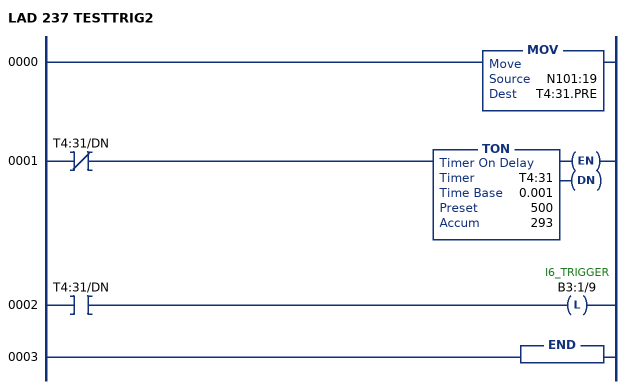
% Rung: 0 %
SOR MOV N101:19 T4:31.PRE EOR
%   N101:19  I6_TRIGTIME  "test trgiger 6 interval" %
% Rung: 1 %
SOR XIO T4:31/DN TON T4:31 0.001 500 293 EOR
% Rung: 2 %
SOR XIC T4:31/DN OTL B3:1/9 EOR
%   B3:1/9  I6_TRIGGER %
% Rung: 3 %
SOR END EOR

LADDER 238 "TESTTRIG3"
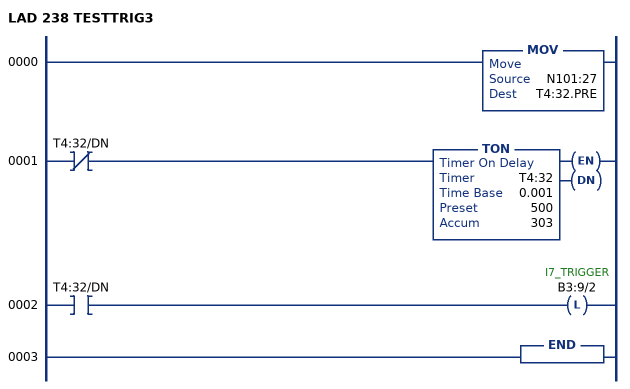
% Rung: 0 %
SOR MOV N101:27 T4:32.PRE EOR
%   N101:27  I7_TRIGTIME %
% Rung: 1 %
SOR XIO T4:32/DN TON T4:32 0.001 500 303 EOR
% Rung: 2 %
SOR XIC T4:32/DN OTL B3:9/2 EOR
%   B3:9/2  I7_TRIGGER %
% Rung: 3 %
SOR END EOR

LADDER 239 "TESTTRIG4"
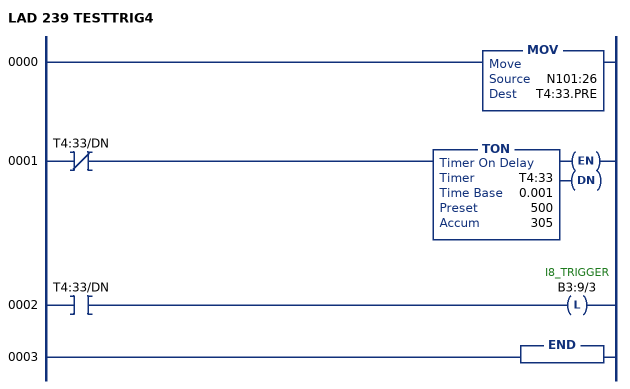
% Rung: 0 %
SOR MOV N101:26 T4:33.PRE EOR
%   N101:26  I8_TRIGTIME %
% Rung: 1 %
SOR XIO T4:33/DN TON T4:33 0.001 500 305 EOR
% Rung: 2 %
SOR XIC T4:33/DN OTL B3:9/3 EOR
%   B3:9/3  I8_TRIGGER %
% Rung: 3 %
SOR END EOR

LADDER 240 "TESTTRIG5"
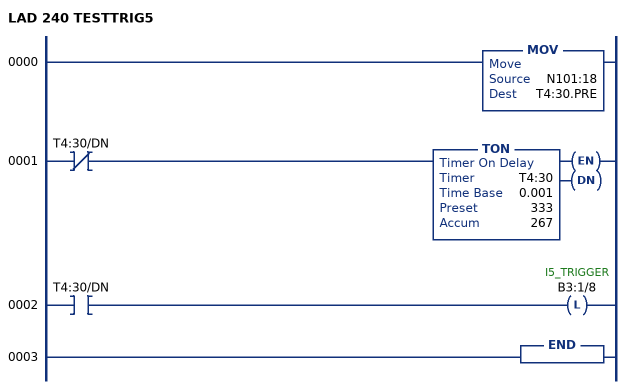
% Rung: 0 %
SOR MOV N101:18 T4:30.PRE EOR
%   N101:18  I5_TRIGTIME  "test trigger 5 interval" %
% Rung: 1 %
SOR XIO T4:30/DN TON T4:30 0.001 333 267 EOR
% Rung: 2 %
SOR XIC T4:30/DN OTL B3:1/8 EOR
%   B3:1/8  I5_TRIGGER %
% Rung: 3 %
SOR END EOR

LADDER 241 "TESTTRIG6"
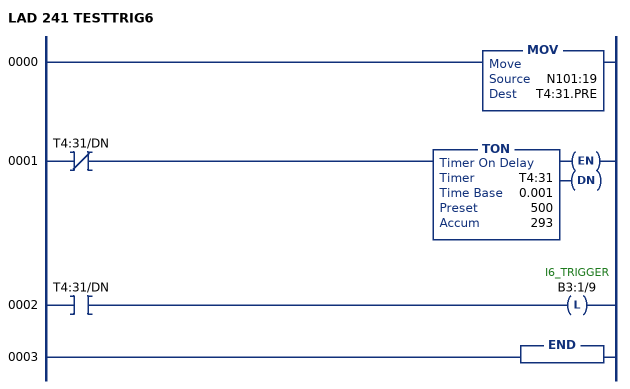
% Rung: 0 %
SOR MOV N101:19 T4:31.PRE EOR
%   N101:19  I6_TRIGTIME  "test trgiger 6 interval" %
% Rung: 1 %
SOR XIO T4:31/DN TON T4:31 0.001 500 293 EOR
% Rung: 2 %
SOR XIC T4:31/DN OTL B3:1/9 EOR
%   B3:1/9  I6_TRIGGER %
% Rung: 3 %
SOR END EOR

LADDER 242 "TESTTRIG7"
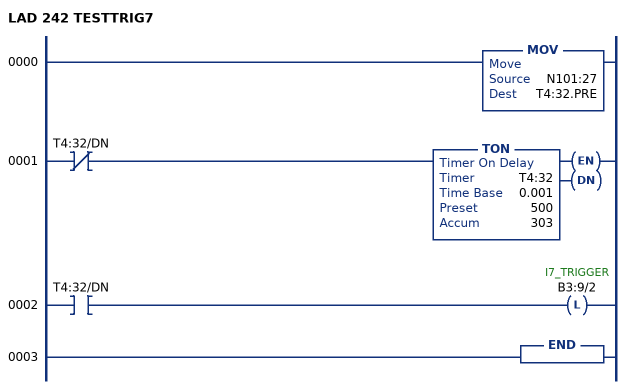
% Rung: 0 %
SOR MOV N101:27 T4:32.PRE EOR
%   N101:27  I7_TRIGTIME %
% Rung: 1 %
SOR XIO T4:32/DN TON T4:32 0.001 500 303 EOR
% Rung: 2 %
SOR XIC T4:32/DN OTL B3:9/2 EOR
%   B3:9/2  I7_TRIGGER %
% Rung: 3 %
SOR END EOR

LADDER 243 "TESTTRIG8"
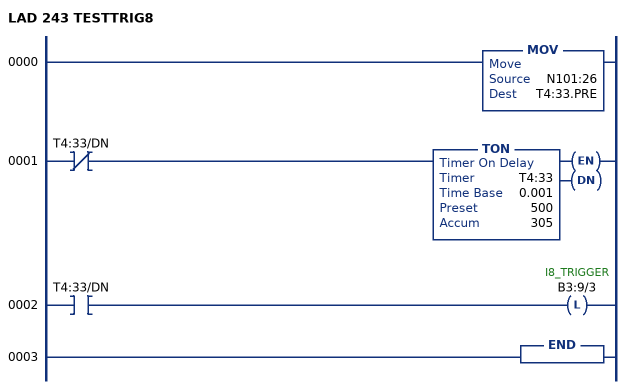
% Rung: 0 %
SOR MOV N101:26 T4:33.PRE EOR
%   N101:26  I8_TRIGTIME %
% Rung: 1 %
SOR XIO T4:33/DN TON T4:33 0.001 500 305 EOR
% Rung: 2 %
SOR XIC T4:33/DN OTL B3:9/3 EOR
%   B3:9/3  I8_TRIGGER %
% Rung: 3 %
SOR END EOR

LADDER 244 "PACKAGER"    % normal %
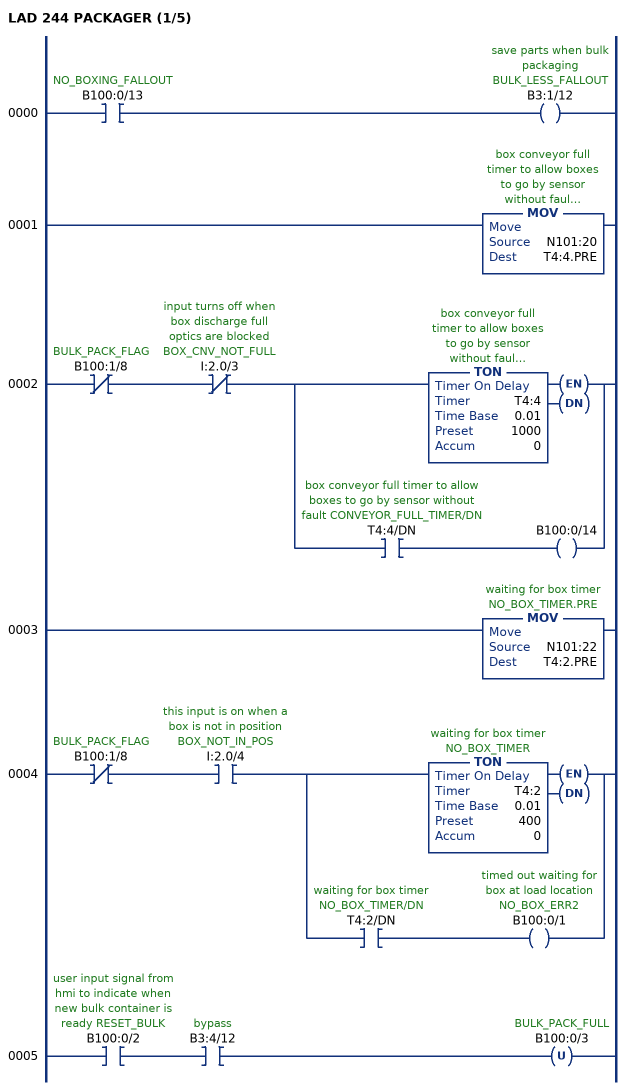
% Rung: 0 %
SOR XIC B100:0/13 OTE B3:1/12 EOR
%   B100:0/13  NO_BOXING_FALLOUT %
%   B3:1/12  BULK_LESS_FALLOUT  "save parts when bulk packaging" %
% Rung: 1 %
SOR MOV N101:20 T4:4.PRE EOR
%   N101:20  CONV_FULL_TIME_LIMIT  "time to allow box to pass box conveyor full sensor without fault" %
%   T4:4  CONVEYOR_FULL_TIMER  "box conveyor full timer to allow boxes to go by sensor without fault" %
% Rung: 2 %
SOR XIO B100:1/8 XIO I:2.0/3 BST TON T4:4 0.01 1000 0 NXB XIC T4:4/DN OTE B100:0/14 BND EOR
%   B100:1/8  BULK_PACK_FLAG %
%   I:2.0/3  BOX_CNV_NOT_FULL  "input turns off when box discharge full optics are blocked" %
%   T4:4  CONVEYOR_FULL_TIMER  "box conveyor full timer to allow boxes to go by sensor without fault" %
% Rung: 3 %
SOR MOV N101:22 T4:2.PRE EOR
%   N101:22  BOX_WAIT_TIME_LIMIT  "the time until waiting for box message in hmi (fault)" %
%   T4:2  NO_BOX_TIMER  "waiting for box timer" %
% Rung: 4 %
SOR XIO B100:1/8 XIC I:2.0/4 BST TON T4:2 0.01 400 0 NXB XIC T4:2/DN OTE B100:0/1 BND EOR
%   B100:1/8  BULK_PACK_FLAG %
%   I:2.0/4  BOX_NOT_IN_POS  "this input is on when a box is not in position" %
%   T4:2  NO_BOX_TIMER  "waiting for box timer" %
%   B100:0/1  NO_BOX_ERR2  "timed out waiting for box at load location" %
% Rung: 5 %
SOR XIC B100:0/2 XIC B3:4/12 OTU B100:0/3 EOR
%   B100:0/2  RESET_BULK  "user input signal from hmi to indicate when new bulk container is ready" %
%   B3:4/12  "bypass" %
%   B100:0/3  BULK_PACK_FULL %

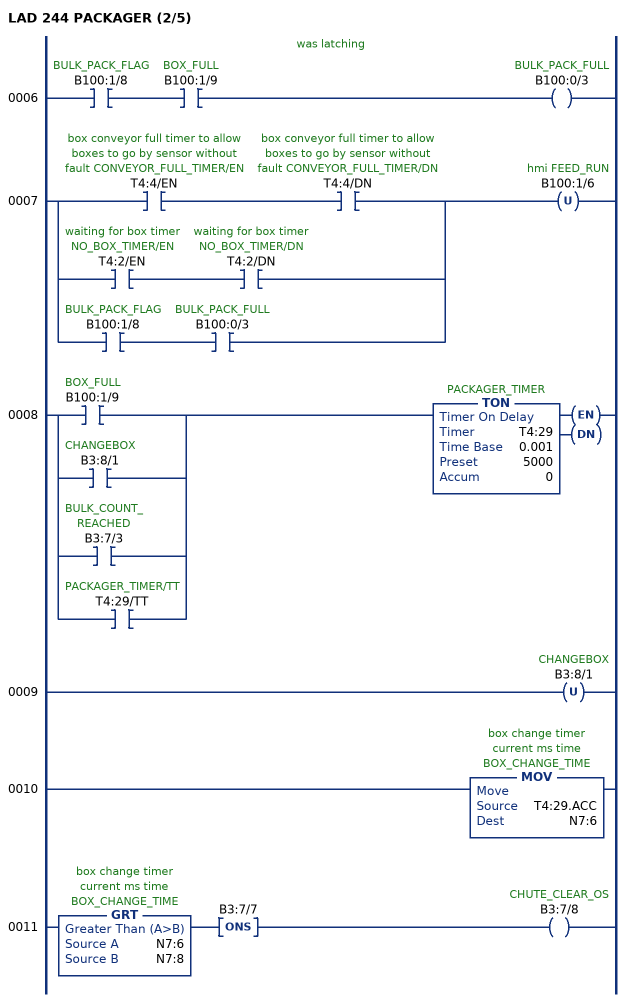
% Rung: 6 %
% was latching %
SOR XIC B100:1/8 XIC B100:1/9 OTE B100:0/3 EOR
%   B100:1/8  BULK_PACK_FLAG %
%   B100:1/9  BOX_FULL %
%   B100:0/3  BULK_PACK_FULL %
% Rung: 7 %
SOR BST XIC T4:4/EN XIC T4:4/DN NXB XIC T4:2/EN XIC T4:2/DN NXB XIC B100:1/8 XIC B100:0/3 BND OTU B100:1/6 EOR
%   T4:4  CONVEYOR_FULL_TIMER  "box conveyor full timer to allow boxes to go by sensor without fault" %
%   T4:2  NO_BOX_TIMER  "waiting for box timer" %
%   B100:1/8  BULK_PACK_FLAG %
%   B100:0/3  BULK_PACK_FULL %
%   B100:1/6  FEED_RUN  "hmi" %
% Rung: 8 %
SOR BST XIC B100:1/9 NXB XIC B3:8/1 NXB XIC B3:7/3 NXB XIC T4:29/TT BND TON T4:29 0.001 5000 0 EOR
%   B100:1/9  BOX_FULL %
%   B3:8/1  CHANGEBOX %
%   B3:7/3  BULK_COUNT_REACHED %
%   T4:29  PACKAGER_TIMER %
% Rung: 9 %
SOR OTU B3:8/1 EOR
%   B3:8/1  CHANGEBOX %
% Rung: 10 %
SOR MOV T4:29.ACC N7:6 EOR
%   T4:29  PACKAGER_TIMER %
%   N7:6  BOX_CHANGE_TIME  "box change timer current ms time" %
% Rung: 11 %
SOR GRT N7:6 N7:8 ONS B3:7/7 OTE B3:7/8 EOR
%   N7:6  BOX_CHANGE_TIME  "box change timer current ms time" %
%   N7:8  CHUTE_CLEAR_TIME %
%   B3:7/8  CHUTE_CLEAR_OS %

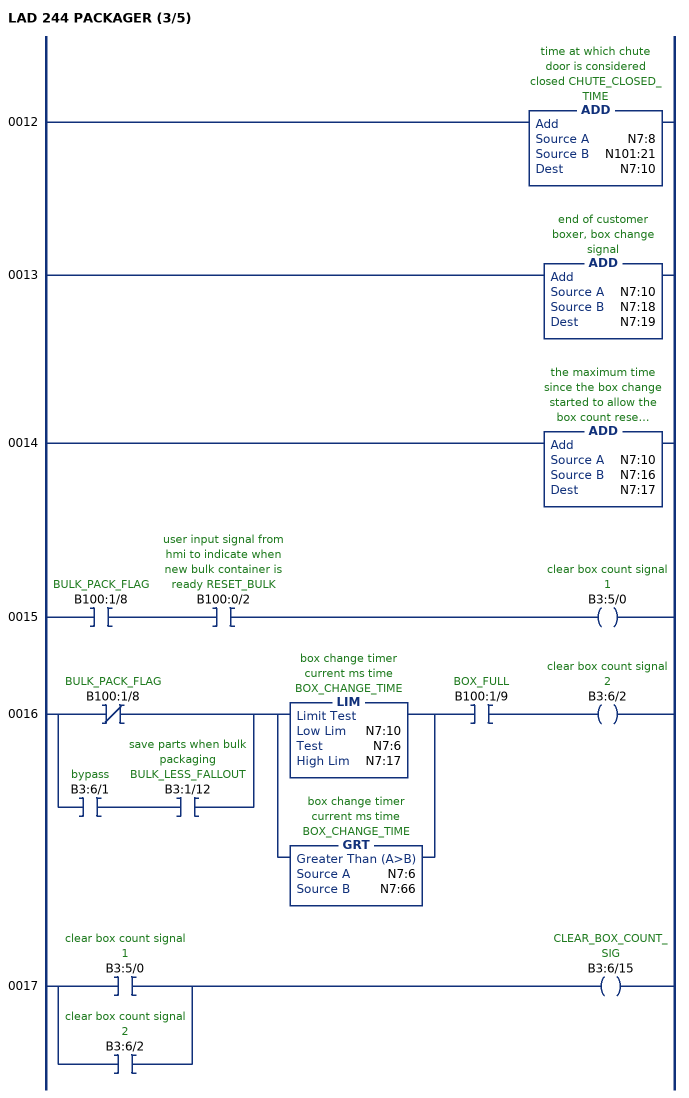
% Rung: 12 %
SOR ADD N7:8 N101:21 N7:10 EOR
%   N7:8  CHUTE_CLEAR_TIME %
%   N101:21  CHUTE_CLOSE_TIME  "ms time required to close chute" %
%   N7:10  CHUTE_CLOSED_TIME  "time at which chute door is considered closed" %
% Rung: 13 %
SOR ADD N7:10 N7:18 N7:19 EOR
%   N7:10  CHUTE_CLOSED_TIME  "time at which chute door is considered closed" %
%   N7:18  CHANGE_BOX_SIG_TIME  "customer boxer change box signal time" %
%   N7:19  "end of customer boxer, box change signal" %
% Rung: 14 %
SOR ADD N7:10 N7:16 N7:17 EOR
%   N7:10  CHUTE_CLOSED_TIME  "time at which chute door is considered closed" %
%   N7:16  RESET_COUNT_SIG_TIME  "maximum length of time to hold box count reset signal on" %
%   N7:17  "the maximum time since the box change started to allow the box count reset signal" %
% Rung: 15 %
SOR XIC B100:1/8 XIC B100:0/2 OTE B3:5/0 EOR
%   B100:1/8  BULK_PACK_FLAG %
%   B100:0/2  RESET_BULK  "user input signal from hmi to indicate when new bulk container is ready" %
%   B3:5/0  "clear box count signal 1" %
% Rung: 16 %
SOR BST XIO B100:1/8 NXB XIC B3:6/1 XIC B3:1/12 BND BST LIM N7:10 N7:6 N7:17 NXB GRT N7:6 N7:66 BND XIC B100:1/9 OTE B3:6/2 EOR
%   B100:1/8  BULK_PACK_FLAG %
%   B3:6/1  "bypass" %
%   B3:1/12  BULK_LESS_FALLOUT  "save parts when bulk packaging" %
%   N7:10  CHUTE_CLOSED_TIME  "time at which chute door is considered closed" %
%   N7:6  BOX_CHANGE_TIME  "box change timer current ms time" %
%   N7:17  "the maximum time since the box change started to allow the box count reset signal" %
%   B100:1/9  BOX_FULL %
%   B3:6/2  "clear box count signal 2" %
% Rung: 17 %
SOR BST XIC B3:5/0 NXB XIC B3:6/2 BND OTE B3:6/15 EOR
%   B3:5/0  "clear box count signal 1" %
%   B3:6/2  "clear box count signal 2" %
%   B3:6/15  CLEAR_BOX_COUNT_SIG %

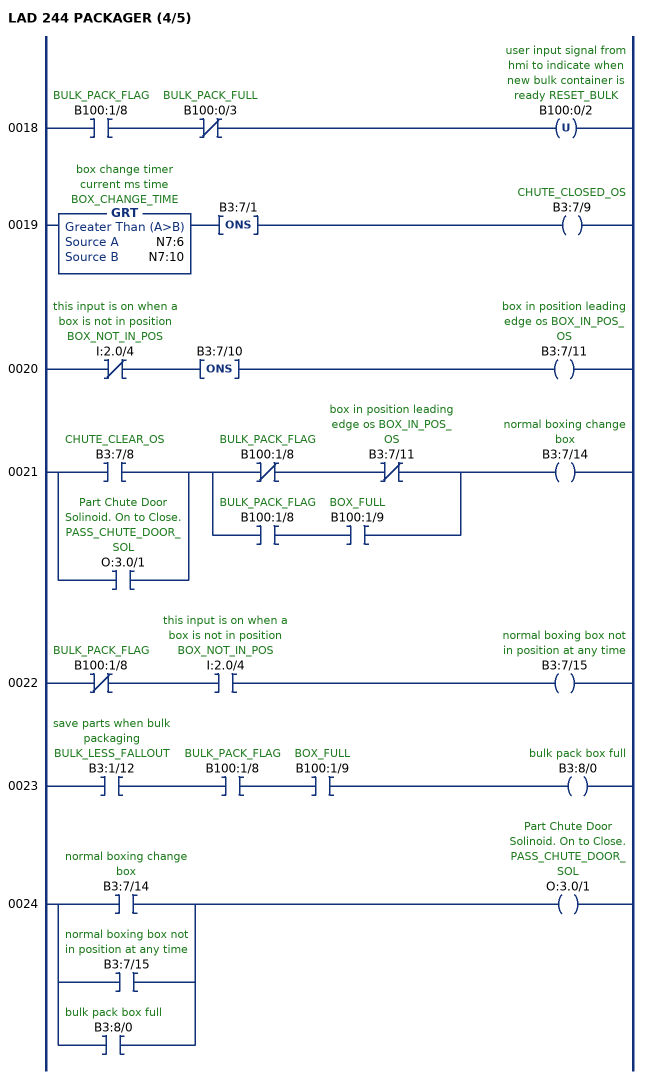
% Rung: 18 %
SOR XIC B100:1/8 XIO B100:0/3 OTU B100:0/2 EOR
%   B100:1/8  BULK_PACK_FLAG %
%   B100:0/3  BULK_PACK_FULL %
%   B100:0/2  RESET_BULK  "user input signal from hmi to indicate when new bulk container is ready" %
% Rung: 19 %
SOR GRT N7:6 N7:10 ONS B3:7/1 OTE B3:7/9 EOR
%   N7:6  BOX_CHANGE_TIME  "box change timer current ms time" %
%   N7:10  CHUTE_CLOSED_TIME  "time at which chute door is considered closed" %
%   B3:7/9  CHUTE_CLOSED_OS %
% Rung: 20 %
SOR XIO I:2.0/4 ONS B3:7/10 OTE B3:7/11 EOR
%   I:2.0/4  BOX_NOT_IN_POS  "this input is on when a box is not in position" %
%   B3:7/11  BOX_IN_POS_OS  "box in position leading edge os" %
% Rung: 21 %
SOR BST XIC B3:7/8 NXB XIC O:3.0/1 BND BST XIO B100:1/8 XIO B3:7/11 NXB XIC B100:1/8 XIC B100:1/9 BND OTE B3:7/14 EOR
%   B3:7/8  CHUTE_CLEAR_OS %
%   O:3.0/1  PASS_CHUTE_DOOR_SOL  "Part Chute Door Solinoid. On to Close." %
%   B100:1/8  BULK_PACK_FLAG %
%   B3:7/11  BOX_IN_POS_OS  "box in position leading edge os" %
%   B100:1/9  BOX_FULL %
%   B3:7/14  "normal boxing change box" %
% Rung: 22 %
SOR XIO B100:1/8 XIC I:2.0/4 OTE B3:7/15 EOR
%   B100:1/8  BULK_PACK_FLAG %
%   I:2.0/4  BOX_NOT_IN_POS  "this input is on when a box is not in position" %
%   B3:7/15  "normal boxing box not in position at any time" %
% Rung: 23 %
SOR XIC B3:1/12 XIC B100:1/8 XIC B100:1/9 OTE B3:8/0 EOR
%   B3:1/12  BULK_LESS_FALLOUT  "save parts when bulk packaging" %
%   B100:1/8  BULK_PACK_FLAG %
%   B100:1/9  BOX_FULL %
%   B3:8/0  "bulk pack box full" %
% Rung: 24 %
SOR BST XIC B3:7/14 NXB XIC B3:7/15 NXB XIC B3:8/0 BND OTE O:3.0/1 EOR
%   B3:7/14  "normal boxing change box" %
%   B3:7/15  "normal boxing box not in position at any time" %
%   B3:8/0  "bulk pack box full" %
%   O:3.0/1  PASS_CHUTE_DOOR_SOL  "Part Chute Door Solinoid. On to Close." %

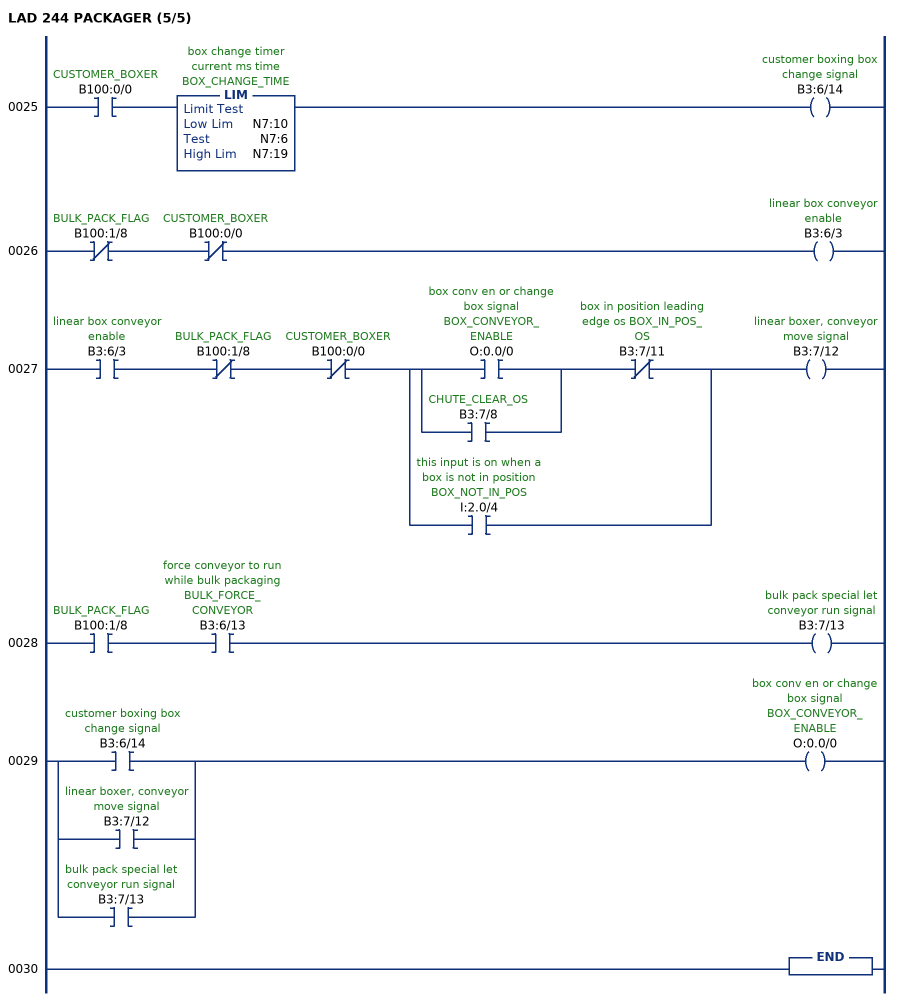
% Rung: 25 %
SOR XIC B100:0/0 LIM N7:10 N7:6 N7:19 OTE B3:6/14 EOR
%   B100:0/0  CUSTOMER_BOXER %
%   N7:10  CHUTE_CLOSED_TIME  "time at which chute door is considered closed" %
%   N7:6  BOX_CHANGE_TIME  "box change timer current ms time" %
%   N7:19  "end of customer boxer, box change signal" %
%   B3:6/14  "customer boxing box change signal" %
% Rung: 26 %
SOR XIO B100:1/8 XIO B100:0/0 OTE B3:6/3 EOR
%   B100:1/8  BULK_PACK_FLAG %
%   B100:0/0  CUSTOMER_BOXER %
%   B3:6/3  "linear box conveyor enable" %
% Rung: 27 %
SOR XIC B3:6/3 XIO B100:1/8 XIO B100:0/0 BST BST XIC O:0.0/0 NXB XIC B3:7/8 BND XIO B3:7/11 NXB XIC I:2.0/4 BND OTE B3:7/12 EOR
%   B3:6/3  "linear box conveyor enable" %
%   B100:1/8  BULK_PACK_FLAG %
%   B100:0/0  CUSTOMER_BOXER %
%   O:0.0/0  BOX_CONVEYOR_ENABLE  "box conv en or change box signal" %
%   B3:7/8  CHUTE_CLEAR_OS %
%   B3:7/11  BOX_IN_POS_OS  "box in position leading edge os" %
%   I:2.0/4  BOX_NOT_IN_POS  "this input is on when a box is not in position" %
%   B3:7/12  "linear boxer, conveyor move signal" %
% Rung: 28 %
SOR XIC B100:1/8 XIC B3:6/13 OTE B3:7/13 EOR
%   B100:1/8  BULK_PACK_FLAG %
%   B3:6/13  BULK_FORCE_CONVEYOR  "force conveyor to run while bulk packaging" %
%   B3:7/13  "bulk pack special let conveyor run signal" %
% Rung: 29 %
SOR BST XIC B3:6/14 NXB XIC B3:7/12 NXB XIC B3:7/13 BND OTE O:0.0/0 EOR
%   B3:6/14  "customer boxing box change signal" %
%   B3:7/12  "linear boxer, conveyor move signal" %
%   B3:7/13  "bulk pack special let conveyor run signal" %
%   O:0.0/0  BOX_CONVEYOR_ENABLE  "box conv en or change box signal" %
% Rung: 30 %
SOR END EOR

LADDER 245 "NO PACKAGE"
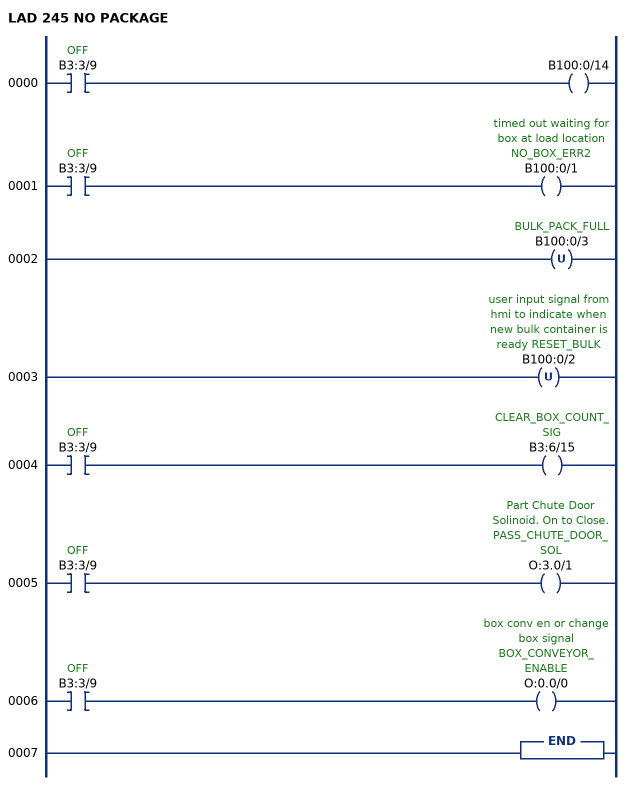
% Rung: 0 %
SOR XIC B3:3/9 OTE B100:0/14 EOR
%   B3:3/9  OFF %
% Rung: 1 %
SOR XIC B3:3/9 OTE B100:0/1 EOR
%   B3:3/9  OFF %
%   B100:0/1  NO_BOX_ERR2  "timed out waiting for box at load location" %
% Rung: 2 %
SOR OTU B100:0/3 EOR
%   B100:0/3  BULK_PACK_FULL %
% Rung: 3 %
SOR OTU B100:0/2 EOR
%   B100:0/2  RESET_BULK  "user input signal from hmi to indicate when new bulk container is ready" %
% Rung: 4 %
SOR XIC B3:3/9 OTE B3:6/15 EOR
%   B3:3/9  OFF %
%   B3:6/15  CLEAR_BOX_COUNT_SIG %
% Rung: 5 %
SOR XIC B3:3/9 OTE O:3.0/1 EOR
%   B3:3/9  OFF %
%   O:3.0/1  PASS_CHUTE_DOOR_SOL  "Part Chute Door Solinoid. On to Close." %
% Rung: 6 %
SOR XIC B3:3/9 OTE O:0.0/0 EOR
%   B3:3/9  OFF %
%   O:0.0/0  BOX_CONVEYOR_ENABLE  "box conv en or change box signal" %
% Rung: 7 %
SOR END EOR

LADDER 246 "RATE1"
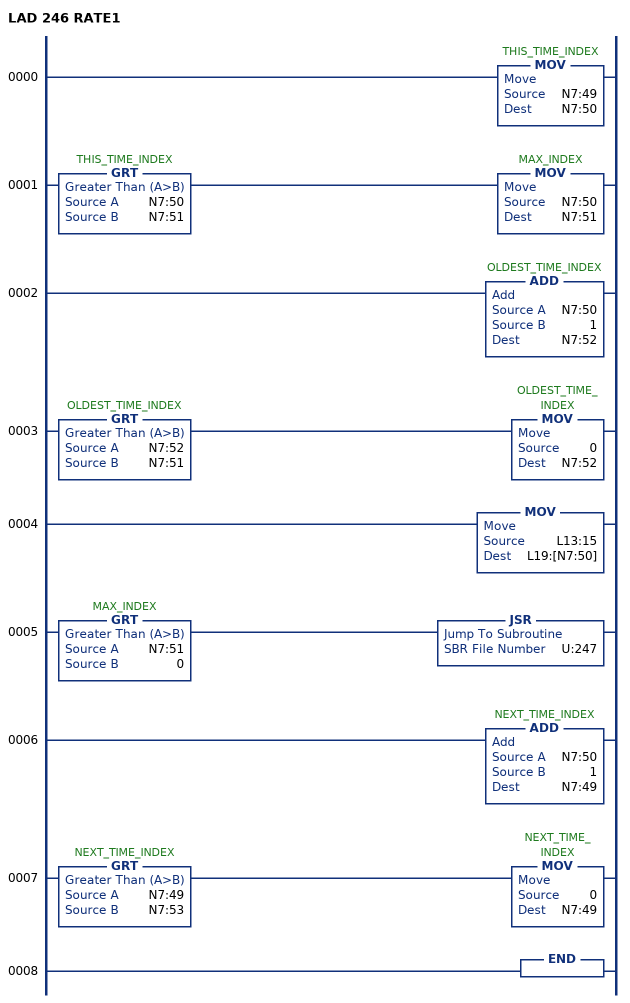
% Rung: 0 %
SOR MOV N7:49 N7:50 EOR
%   N7:49  NEXT_TIME_INDEX %
%   N7:50  THIS_TIME_INDEX %
% Rung: 1 %
SOR GRT N7:50 N7:51 MOV N7:50 N7:51 EOR
%   N7:50  THIS_TIME_INDEX %
%   N7:51  MAX_INDEX %
% Rung: 2 %
SOR ADD N7:50 1 N7:52 EOR
%   N7:50  THIS_TIME_INDEX %
%   N7:52  OLDEST_TIME_INDEX %
% Rung: 3 %
SOR GRT N7:52 N7:51 MOV 0 N7:52 EOR
%   N7:52  OLDEST_TIME_INDEX %
%   N7:51  MAX_INDEX %
% Rung: 4 %
SOR MOV L13:15 L19:[N7:50] EOR
%   L13:15  THE_TIME %
%   N7:50  THIS_TIME_INDEX %
% Rung: 5 %
SOR GRT N7:51 0 JSR U:247 EOR
%   N7:51  MAX_INDEX %
% Rung: 6 %
SOR ADD N7:50 1 N7:49 EOR
%   N7:50  THIS_TIME_INDEX %
%   N7:49  NEXT_TIME_INDEX %
% Rung: 7 %
SOR GRT N7:49 N7:53 MOV 0 N7:49 EOR
%   N7:49  NEXT_TIME_INDEX %
%   N7:53  UPPER_INDEX_LIMIT %
% Rung: 8 %
SOR END EOR

LADDER 247 "RATE2"
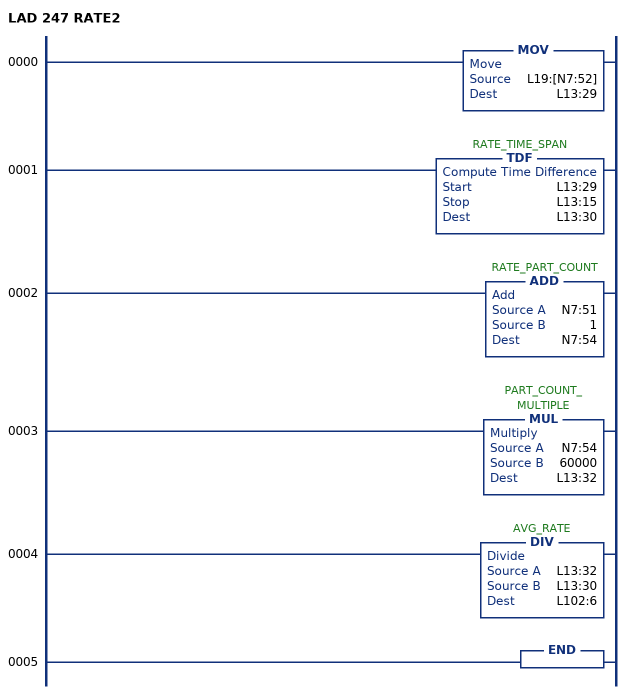
% Rung: 0 %
SOR MOV L19:[N7:52] L13:29 EOR
%   N7:52  OLDEST_TIME_INDEX %
% Rung: 1 %
SOR TDF L13:29 L13:15 L13:30 EOR
%   L13:15  THE_TIME %
%   L13:30  RATE_TIME_SPAN %
% Rung: 2 %
SOR ADD N7:51 1 N7:54 EOR
%   N7:51  MAX_INDEX %
%   N7:54  RATE_PART_COUNT %
% Rung: 3 %
SOR MUL N7:54 60000 L13:32 EOR
%   N7:54  RATE_PART_COUNT %
%   L13:32  PART_COUNT_MULTIPLE %
% Rung: 4 %
SOR DIV L13:32 L13:30 L102:6 EOR
%   L13:32  PART_COUNT_MULTIPLE %
%   L13:30  RATE_TIME_SPAN %
%   L102:6  AVG_RATE %
% Rung: 5 %
SOR END EOR

LADDER 248 "RESET RATE"
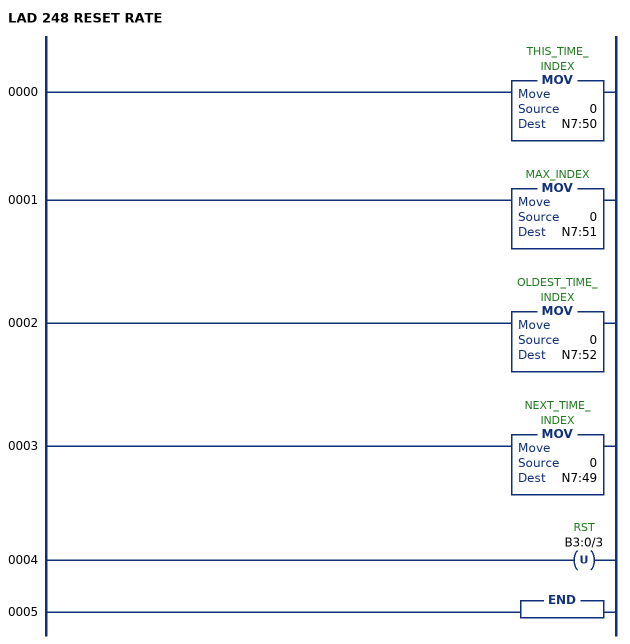
% Rung: 0 %
SOR MOV 0 N7:50 EOR
%   N7:50  THIS_TIME_INDEX %
% Rung: 1 %
SOR MOV 0 N7:51 EOR
%   N7:51  MAX_INDEX %
% Rung: 2 %
SOR MOV 0 N7:52 EOR
%   N7:52  OLDEST_TIME_INDEX %
% Rung: 3 %
SOR MOV 0 N7:49 EOR
%   N7:49  NEXT_TIME_INDEX %
% Rung: 4 %
SOR OTU B3:0/3 EOR
%   B3:0/3  RST %
% Rung: 5 %
SOR END EOR

LADDER 249 "NP STOP"    % stop on no good %
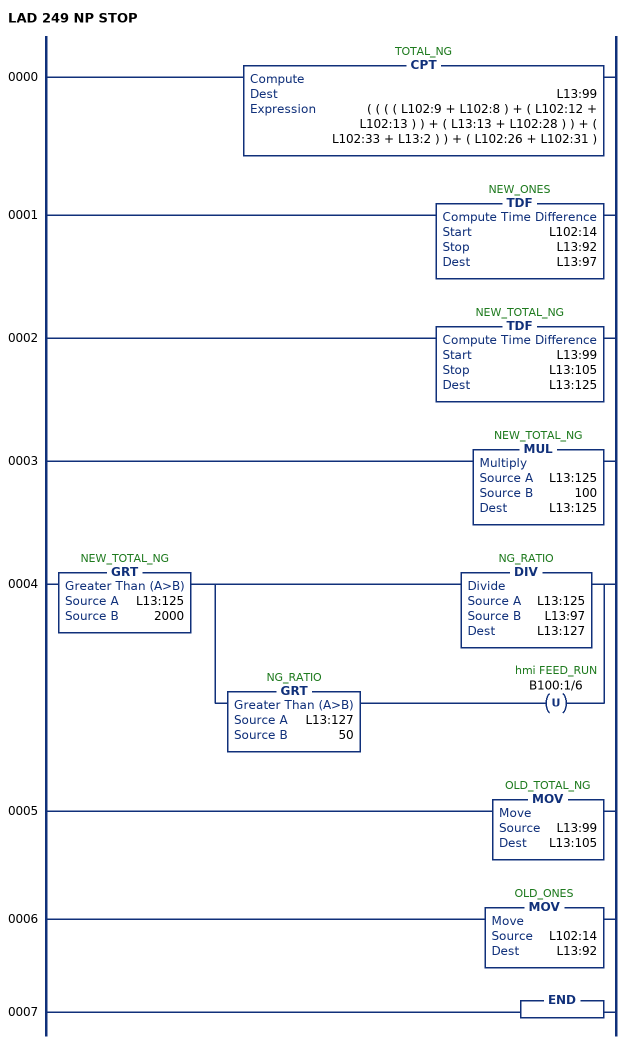
% Rung: 0 %
SOR CPT L13:99 " ( ( ( ( L102:9 + L102:8 ) + ( L102:12 + L102:13 ) ) + ( L13:13 + L102:28 ) ) + ( L102:33 + L13:2 ) ) + ( L102:26 + L102:31 ) " EOR
%   L13:99  TOTAL_NG %
%   L102:9  "too wide bottom" %
%   L102:8  "too close bottom" %
%   L102:12  "too close top count" %
%   L102:13  "too wide top count" %
%   L102:28  I1_I5_SKIPPEDCOUNT %
%   L102:33  I6_SKIPPEDCOUNT %
%   L102:26  I1_I5_FAIL_COUNT %
%   L102:31  I6_FAIL_COUNT %
% Rung: 1 %
SOR TDF L102:14 L13:92 L13:97 EOR
%   L102:14  ONES %
%   L13:92  OLD_ONES %
%   L13:97  NEW_ONES %
% Rung: 2 %
SOR TDF L13:99 L13:105 L13:125 EOR
%   L13:99  TOTAL_NG %
%   L13:105  OLD_TOTAL_NG %
%   L13:125  NEW_TOTAL_NG %
% Rung: 3 %
SOR MUL L13:125 100 L13:125 EOR
%   L13:125  NEW_TOTAL_NG %
% Rung: 4 %
SOR GRT L13:125 2000 BST DIV L13:125 L13:97 L13:127 NXB GRT L13:127 50 OTU B100:1/6 BND EOR
%   L13:125  NEW_TOTAL_NG %
%   L13:97  NEW_ONES %
%   L13:127  NG_RATIO %
%   B100:1/6  FEED_RUN  "hmi" %
% Rung: 5 %
SOR MOV L13:99 L13:105 EOR
%   L13:99  TOTAL_NG %
%   L13:105  OLD_TOTAL_NG %
% Rung: 6 %
SOR MOV L102:14 L13:92 EOR
%   L102:14  ONES %
%   L13:92  OLD_ONES %
% Rung: 7 %
SOR END EOR

LADDER 250 "SPEED BOT"    % high speed %
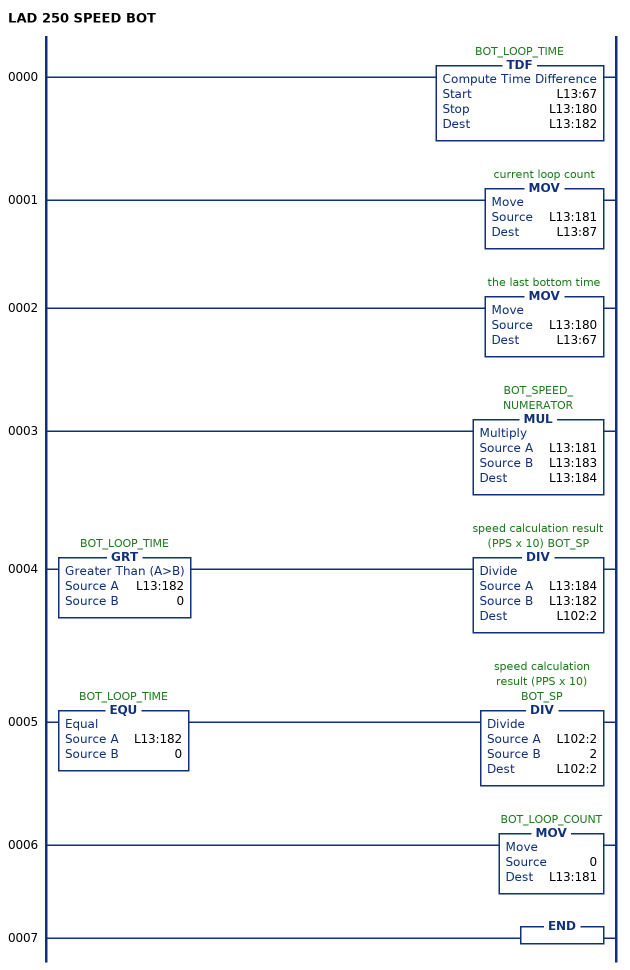
% Rung: 0 %
SOR TDF L13:67 L13:180 L13:182 EOR
%   L13:67  "the last bottom time" %
%   L13:180  BOT_THIS_TIME  "rtc bot belt movement event time" %
%   L13:182  BOT_LOOP_TIME %
% Rung: 1 %
SOR MOV L13:181 L13:87 EOR
%   L13:181  BOT_LOOP_COUNT %
%   L13:87  "current loop count" %
% Rung: 2 %
SOR MOV L13:180 L13:67 EOR
%   L13:180  BOT_THIS_TIME  "rtc bot belt movement event time" %
%   L13:67  "the last bottom time" %
% Rung: 3 %
SOR MUL L13:181 L13:183 L13:184 EOR
%   L13:181  BOT_LOOP_COUNT %
%   L13:183  TKS_PER_SECOND %
%   L13:184  BOT_SPEED_NUMERATOR %
% Rung: 4 %
SOR GRT L13:182 0 DIV L13:184 L13:182 L102:2 EOR
%   L13:182  BOT_LOOP_TIME %
%   L13:184  BOT_SPEED_NUMERATOR %
%   L102:2  BOT_SP  "speed calculation result (PPS x 10)" %
% Rung: 5 %
SOR EQU L13:182 0 DIV L102:2 2 L102:2 EOR
%   L13:182  BOT_LOOP_TIME %
%   L102:2  BOT_SP  "speed calculation result (PPS x 10)" %
% Rung: 6 %
SOR MOV 0 L13:181 EOR
%   L13:181  BOT_LOOP_COUNT %
% Rung: 7 %
SOR END EOR

LADDER 251 "SPEED TOP"    % high speed %
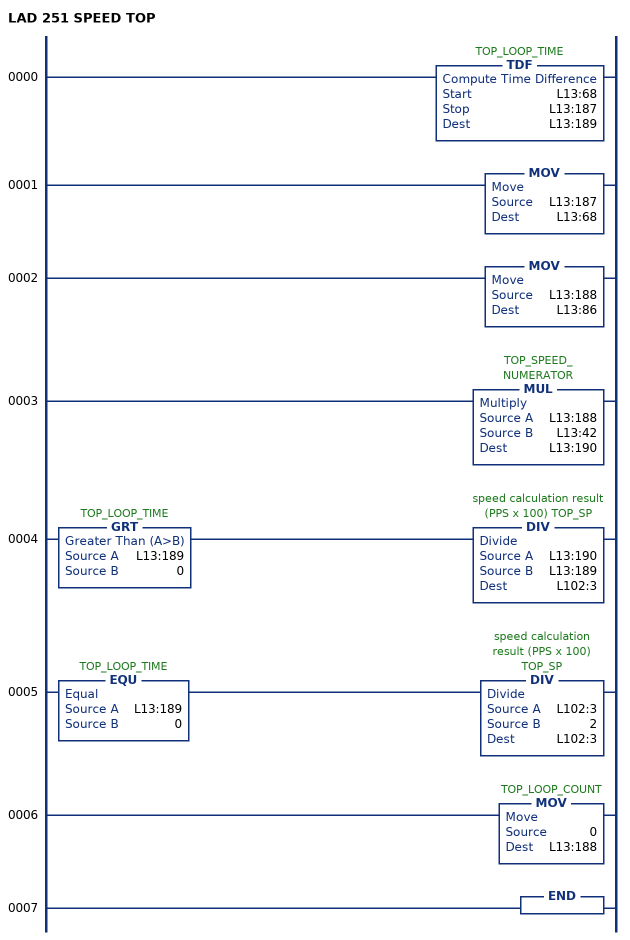
% Rung: 0 %
SOR TDF L13:68 L13:187 L13:189 EOR
%   L13:187  TOP_THIS_TIME  "rtc top belt movement event time" %
%   L13:189  TOP_LOOP_TIME %
% Rung: 1 %
SOR MOV L13:187 L13:68 EOR
%   L13:187  TOP_THIS_TIME  "rtc top belt movement event time" %
% Rung: 2 %
SOR MOV L13:188 L13:86 EOR
%   L13:188  TOP_LOOP_COUNT %
% Rung: 3 %
SOR MUL L13:188 L13:42 L13:190 EOR
%   L13:188  TOP_LOOP_COUNT %
%   L13:190  TOP_SPEED_NUMERATOR %
% Rung: 4 %
SOR GRT L13:189 0 DIV L13:190 L13:189 L102:3 EOR
%   L13:189  TOP_LOOP_TIME %
%   L13:190  TOP_SPEED_NUMERATOR %
%   L102:3  TOP_SP  "speed calculation result (PPS x 100)" %
% Rung: 5 %
SOR EQU L13:189 0 DIV L102:3 2 L102:3 EOR
%   L13:189  TOP_LOOP_TIME %
%   L102:3  TOP_SP  "speed calculation result (PPS x 100)" %
% Rung: 6 %
SOR MOV 0 L13:188 EOR
%   L13:188  TOP_LOOP_COUNT %
% Rung: 7 %
SOR END EOR

LADDER 252 "P BOT"    % high speed %
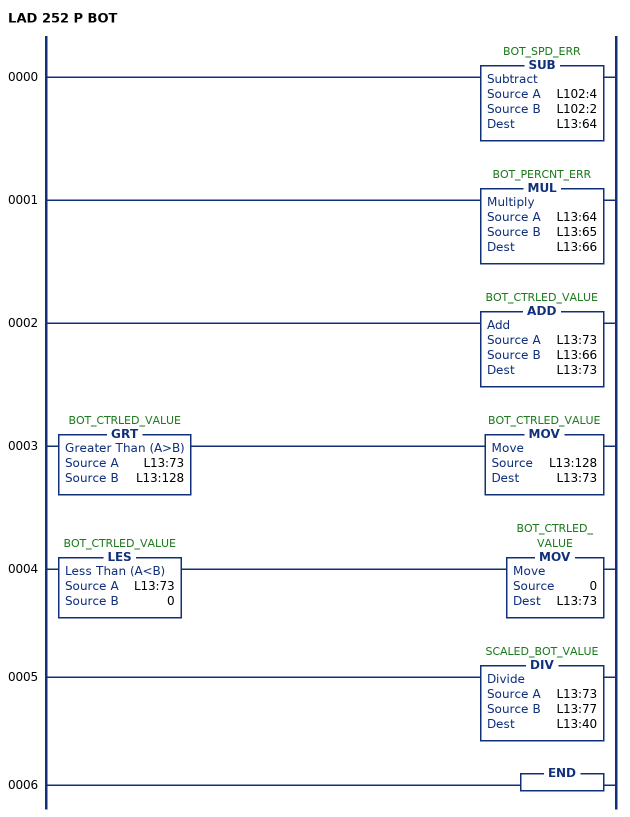
% Rung: 0 %
SOR SUB L102:4 L102:2 L13:64 EOR
%   L102:4  BOT_SPD_SETPOINT %
%   L102:2  BOT_SP  "speed calculation result (PPS x 10)" %
%   L13:64  BOT_SPD_ERR %
% Rung: 1 %
SOR MUL L13:64 L13:65 L13:66 EOR
%   L13:64  BOT_SPD_ERR %
%   L13:65  POS5SHIFT %
%   L13:66  BOT_PERCNT_ERR %
% Rung: 2 %
SOR ADD L13:73 L13:66 L13:73 EOR
%   L13:73  BOT_CTRLED_VALUE %
%   L13:66  BOT_PERCNT_ERR %
% Rung: 3 %
SOR GRT L13:73 L13:128 MOV L13:128 L13:73 EOR
%   L13:73  BOT_CTRLED_VALUE %
%   L13:128  "how much top has shifted since measurment" %
% Rung: 4 %
SOR LES L13:73 0 MOV 0 L13:73 EOR
%   L13:73  BOT_CTRLED_VALUE %
% Rung: 5 %
SOR DIV L13:73 L13:77 L13:40 EOR
%   L13:73  BOT_CTRLED_VALUE %
%   L13:40  SCALED_BOT_VALUE %
% Rung: 6 %
SOR END EOR

LADDER 253 "P TOP"    % high speed %
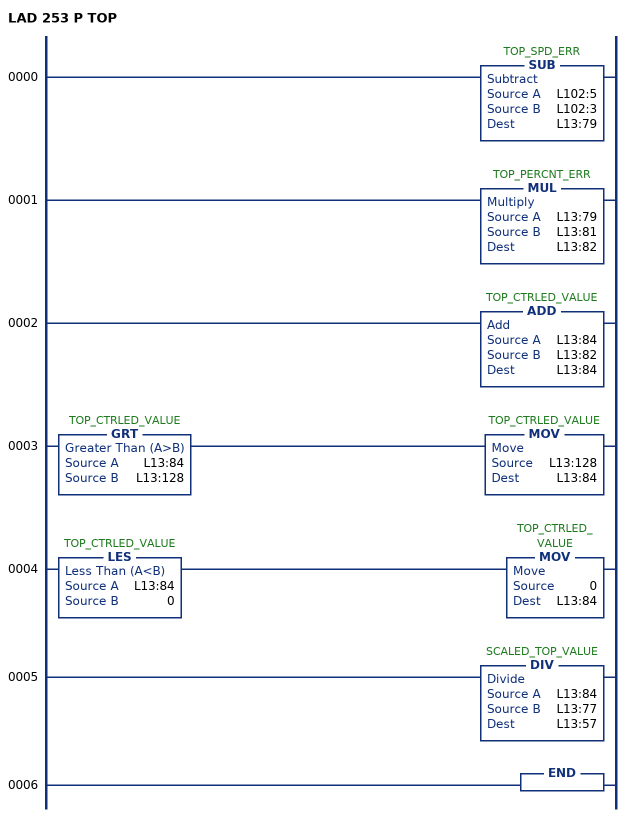
% Rung: 0 %
SOR SUB L102:5 L102:3 L13:79 EOR
%   L102:5  TOP_SPD_SETPOINT %
%   L102:3  TOP_SP  "speed calculation result (PPS x 100)" %
%   L13:79  TOP_SPD_ERR %
% Rung: 1 %
SOR MUL L13:79 L13:81 L13:82 EOR
%   L13:79  TOP_SPD_ERR %
%   L13:81  TOP_FDBK_RATIO %
%   L13:82  TOP_PERCNT_ERR %
% Rung: 2 %
SOR ADD L13:84 L13:82 L13:84 EOR
%   L13:84  TOP_CTRLED_VALUE %
%   L13:82  TOP_PERCNT_ERR %
% Rung: 3 %
SOR GRT L13:84 L13:128 MOV L13:128 L13:84 EOR
%   L13:84  TOP_CTRLED_VALUE %
%   L13:128  "how much top has shifted since measurment" %
% Rung: 4 %
SOR LES L13:84 0 MOV 0 L13:84 EOR
%   L13:84  TOP_CTRLED_VALUE %
% Rung: 5 %
SOR DIV L13:84 L13:77 L13:57 EOR
%   L13:84  TOP_CTRLED_VALUE %
%   L13:57  SCALED_TOP_VALUE %
% Rung: 6 %
SOR END EOR

LADDER 254 "TOTALCOUNT"
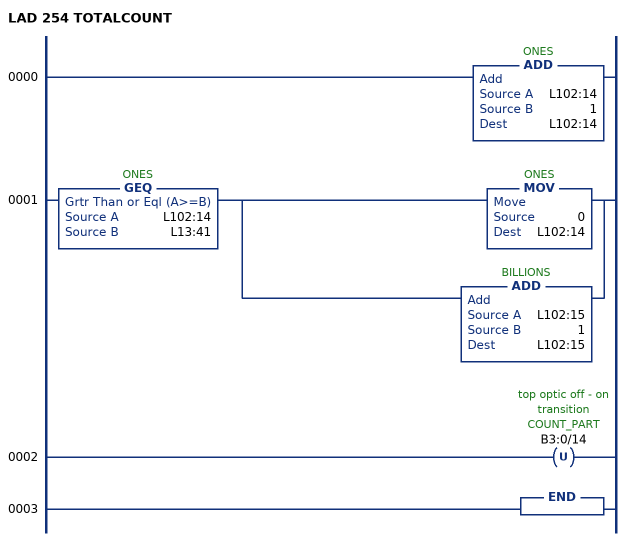
% Rung: 0 %
SOR ADD L102:14 1 L102:14 EOR
%   L102:14  ONES %
% Rung: 1 %
SOR GEQ L102:14 L13:41 BST MOV 0 L102:14 NXB ADD L102:15 1 L102:15 BND EOR
%   L102:14  ONES %
%   L13:41  "skipped count change in the last 3 seconds" %
%   L102:15  BILLIONS %
% Rung: 2 %
SOR OTU B3:0/14 EOR
%   B3:0/14  COUNT_PART  "top optic off - on transition" %
% Rung: 3 %
SOR END EOR

LADDER 255 "SAVED"
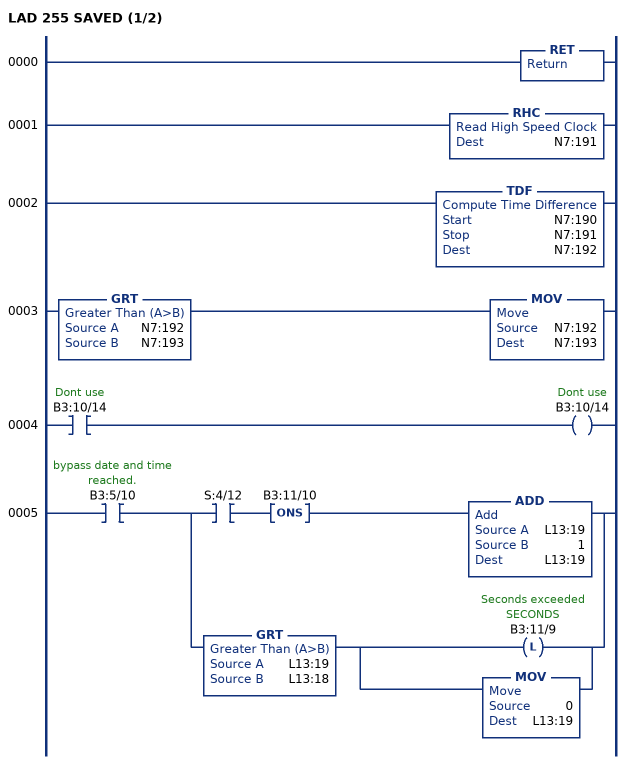
% Rung: 0 %
SOR RET EOR
% Rung: 1 %
SOR RHC N7:191 EOR
% Rung: 2 %
SOR TDF N7:190 N7:191 N7:192 EOR
% Rung: 3 %
SOR GRT N7:192 N7:193 MOV N7:192 N7:193 EOR
% Rung: 4 %
SOR XIC B3:10/14 OTE B3:10/14 EOR
%   B3:10/14  "Dont use" %
% Rung: 5 %
SOR XIC B3:5/10 BST XIC S:4/12 ONS B3:11/10 ADD L13:19 1 L13:19 NXB GRT L13:19 L13:18 BST OTL B3:11/9 NXB MOV 0 L13:19 BND BND EOR
%   B3:5/10  "bypass date and time reached." %
%   L13:18  MAX %
%   B3:11/9  SECONDS  "Seconds exceeded" %

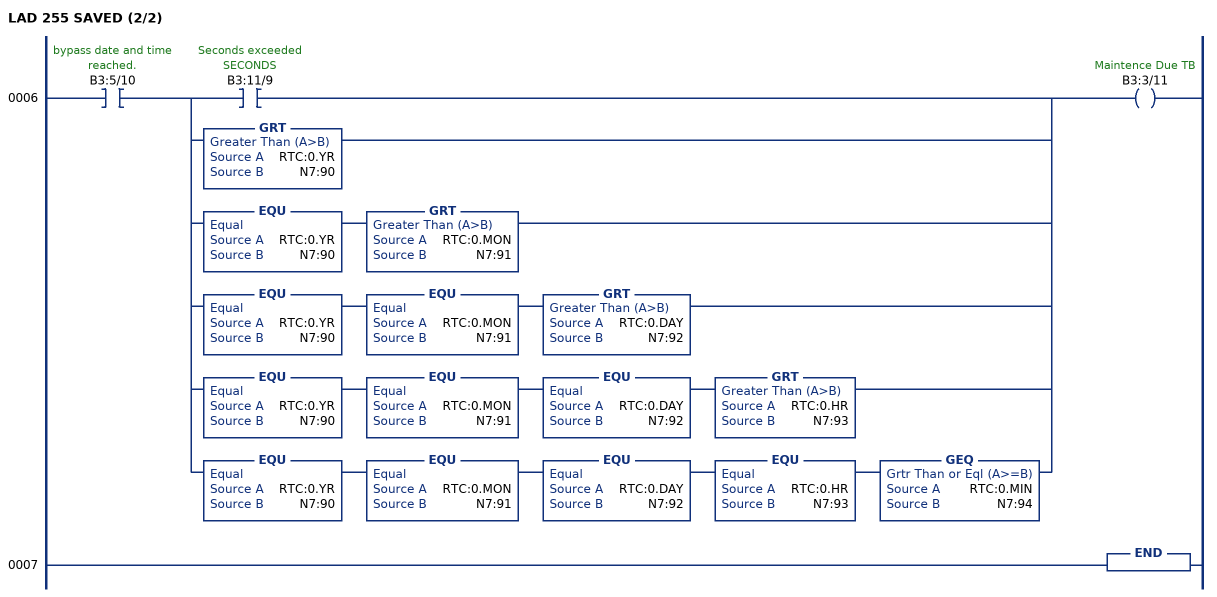
% Rung: 6 %
SOR XIC B3:5/10 BST XIC B3:11/9 NXB GRT RTC:0.YR N7:90 NXB EQU RTC:0.YR N7:90 GRT RTC:0.MON N7:91 NXB EQU RTC:0.YR N7:90 EQU RTC:0.MON N7:91 GRT RTC:0.DAY N7:92 NXB EQU RTC:0.YR N7:90 EQU RTC:0.MON N7:91 EQU RTC:0.DAY N7:92 GRT RTC:0.HR N7:93 NXB EQU RTC:0.YR N7:90 EQU RTC:0.MON N7:91 EQU RTC:0.DAY N7:92 EQU RTC:0.HR N7:93 GEQ RTC:0.MIN N7:94 BND OTE B3:3/11 EOR
%   B3:5/10  "bypass date and time reached." %
%   B3:11/9  SECONDS  "Seconds exceeded" %
%   N7:90  RTC %
%   B3:3/11  TB  "Maintence Due" %
% Rung: 7 %
SOR END EOR

OTHER DOCUMENTED ADDRESSES
  B3:10/3  "bypass"
  B3:11/5  "bypass"
  B3:11/6  "bypass"
  B3:11/7  "bypass"
  B3:11/8  "was jump to inspection #2"
  B3:11/11  "was jump to inspection #3"
  B3:11/12  "was jump to inspection #4"
  B41:0  TOP_OK_3
  B189:0/0  "change box"
  B189:0/9  "override boxing ok or not full signal"
  B189:0/11  "HMI force door close"
  B196:1/0  "Chute door is closed"
  B196:1/1  "control chute door"
  B196:1/13  "force box conveyor on"
  B196:3/0  "for hmi to continue production unlatched by hmi"
  HSC:0.0  "top"
  HSC:0.3/6  "Underflow interrupt"
  HSC:0.3/7  "Overflow interrupt"
  HSC:1.0  "bot"
  HSC:1.3/6  "Underflow interrupt"
  HSC:1.3/7  "Overflow interrupt"
  I:0.0/0  "Encoder Signal "A""
  I:0.0/1  "Encoder Signal "B""
  I:0.0/4  "Encoder Signal "A""
  I:0.0/5  "Encoder Signal "B""
  I:0.1/4  "not used"
  I:0.1/5  "not used"
  I:0.1/6  "not used"
  I:0.1/7  "not used"
  I:0.1/8  "not used"
  I:0.1/9  "not used"
  I:0.1/10  "not used"
  I:0.1/11  "not used"
  I:0.1/12  "not used"
  I:0.1/13  "not used"
  I:0.1/14  "not used"
  I:0.1/15  "not used"
  I:0.2  "not used"
  I:0.2/3  "Packaging Conveyor full"
  I:0.2/4  "Packaging Conveyor Box in Position"
  I:0.3  "not used"
  I:0.4  "Spare Analog Input 1"
  I:0.5  "Spare Analog Input 2"
  I:0.6  "Spare Analog Input 3"
  I:2.0/0  FRONT_ESTOP
  I:2.0/1  REAR_ESTOP
  I:2.0/8  FRONT_DOOR  "front door signal ce models only"
  I:2.0/9  REAR_DOOR  "rear door signal ce models only"
  I:2.0/11  "spare"
  L23:19  TOP_OPT_FAIL_CT
  L23:34  AIR_PRESSURE_FAULT
  L28:0  INS_1_TIME
  L29:0  INS_1_POS
  L30:0  INS_5_TIME
  L31:0  INS_5_POS
  L32:0  INS_6_TIME
  L33:0  INS_6_POS
  L192:1  BOT_LAST_TIME  "rtc bot belt previous movement event time"
  L192:2  BOT_CYCLE_TIME  "rtc bot belt time between events"
  L192:7  FROM_REAL  "distance from real part signal at optic location"
  L192:8  FROM_TRACKED  "distance from tracked part signal at optic location"
  L192:16  TOP_LAST_TIME  "rtc top belt previous movement event time"
  L192:17  TOP_CYCLE_TIME  "rtc top belt time between events"
  L199:5  ACQTM51
  L199:6  ACQTM52
  L199:7  ACQTM53
  L199:9  "ones"
  L199:10  "billions"
  L199:13  DUMP_LONG
  L199:15  ACQTM11
  L199:16  ACQTM12
  L199:17  ACQTM13
  L199:20  RESULTTM1
  L199:22  CLEARTIME5COUNT
  L199:23  CLEARTIME6COUNT
  L199:24  ACQTM61
  L199:25  ACQTM62
  L199:26  ACQTM63
  L199:27  TMSINCETRIG1
  L199:29  TMSINCETRIG5
  L199:30  TMSINCETRIG6
  L199:31  CLEARTIME1COUNT
  L199:32  RESULTTM5
  L199:33  RESULTTM6
  L199:34  MAXACQTM1
  L199:36  MAXACQTM6
  N7:9  TOP_GOOD3_START_WORD
  N101:1  I2_TRIG_LOC
  N101:2  I3_TRIG_LOC
  N101:3  I4_TRIG_LOC
  O:0.0/1  "spare"
  O:0.0/11  "Spare"
  O:0.0/12  "not used"
  O:0.0/13  "not used"
  O:0.0/14  "not used"
  O:0.0/15  "not used"
  O:0.1  "not used"
  O:0.2  "not used"
  O:0.3  "not used"
  O:0.5  "spare analog output"
  O:3.0/0  "spare"
  O:3.0/2  "spare"
  O:3.0/3  "light curtain range selection /* needed? */"
  O:3.0/7  "door unlocks on CE models"
  O:3.0/8  "Light?"
  PFILE:6  "check for part jams"
  PFILE:10  "Bottom belt HSC"
  PFILE:12  "Top belt HSC"
  Q2:55  END_OF_MAIN
  Q5:94  END_OF_BELTS
  T20:0  "Trigger On Time"
  TOP_OPTIC_LO  
  U:3  TEST
  U:9  "slow data"
  U:24  "check skipped fail rate"
  U:28  "faults"
  U:29  "speed"
  U:30  "count"
  U:31  "rate calc"
  U:32  "boxer"
  U:33  "bulk pack"
  U:34  "customer boxing unit signals"
  U:35  "cleanup"

REVISION NOTES
  13: updated count reset
  14: added io moduals
  15: multiple steps toward new hmi integration
  21: test
  27: fix error if bulk pack and no boxing fallout were on

DATA TABLE (non-zero values as saved)
DATA B3
% B3:0 % 0XA034 0X0160 0X4001 0X5109 0X0EF3 0X0D24 0X0DB0 0X0421 0X5F80 0X2330
% B3:10 % 0X21F4 0X000E 0X2000 0X0000 0X0000 0X0000 0X0000 0X0000 0X0000 0X0000
% B3:50 % 0X0001 0X0000 0X0000 0X0000 0X0000 0X0000 0X0000 0X0000 0X0000 0X0000
DATA T4
% .PRE .ACC %
% T4:0 % 0 3
% T4:1 % 150 0
% T4:2 % 400 0
% T4:3 % 500 307
% T4:4 % 1000 0
% T4:5 % 5 5
% T4:6 % 10 32766
% T4:7 % 666 0
% T4:8 % 20 12
% T4:9 % 50 8
% T4:10 % 200 200
% T4:11 % 111 0
% T4:12 % 40 40
% T4:13 % 250 0
% T4:14 % 666 0
% T4:15 % 1000 1000
% T4:16 % 400 0
% T4:17 % 100 34
% T4:18 % 5 0
% T4:19 % 300 0
% T4:20 % 200 0
% T4:21 % 200 0
% T4:22 % 200 0
% T4:23 % 250 0
% T4:24 % 666 0
% T4:25 % 666 0
% T4:26 % 666 0
% T4:27 % 250 0
% T4:28 % 250 0
% T4:29 % 5000 0
% T4:30 % 333 267
% T4:31 % 500 293
% T4:32 % 500 303
% T4:33 % 500 305
DATA C5
% .PRE .ACC %
% C5:0 % 32766 0
DATA R6
% .LEN .POS %
% R6:0 % 1250 0
% R6:1 % 1250 0
% R6:2 % 1050 0
% R6:3 % 1050 0
% R6:4 % 1250 0
% R6:5 % 1250 0
% R6:6 % 1713 0
% R6:7 % 1024 0
% R6:8 % 1024 0
% R6:9 % 3 0
% R6:10 % 2048 0
% R6:11 % 2048 0
% R6:12 % 10 0
% R6:13 % 10 0
% R6:14 % 10 0
% R6:15 % 10 0
% R6:16 % 1713 0
% R6:17 % 2048 0
% R6:18 % 2048 0
% R6:19 % 10 0
DATA N7
% N7:0 % 17247 3 1015 166 3 202 0 0 500 43
% N7:10 % 1000 0 0 2 20 20 1000 2000 50 1050
% N7:20 % 0 598 10 13 208 46 0 0 150 250
% N7:30 % 666 0 150 0 48 1231 77 9 0 9
% N7:40 % 48 12 0 12 32767 1248 222 256 1636 3
% N7:50 % 2 2 0 16 3 1024 0 0 32766 0
% N7:60 % 1713 2048 2048 984 1034 1024 4999 5 400 400
% N7:70 % 100 200 300 400 90 190 290 390 0 0
% N7:80 % 0 0 1256 1263 1278 1288 9 13 0 0
% N7:90 % 2011 4 4 12 1 9 13 222 222 12
% N7:100 % 1003 90 110 100 175 25 0 0 0 0
% N7:190 % 18705 17572 55 88 0 0 0 0 0 0
DATA F8
% F8:0 % 6
DATA L13
% L13:0 % 12165 115601 0 34982 170009
% L13:5 % 5 2 5 131249 2
% L13:10 % 2 3332502 30832 15 90
% L13:15 % 1189265907 -2147483648 2147483647 2147483647 82058
% L13:20 % 20821667 1941975217 777 33055 100
% L13:25 % 5304 2236 2815602 2 1188992105
% L13:30 % 273449 5 180000 1188692964 444
% L13:35 % 1 624336 0 0 0
% L13:40 % 30019 1000000000 1000000 1188692931 1189189992
% L13:45 % 1189191387 150 0 33 20590662
% L13:50 % 75915 294744 1189189964 0 0
% L13:55 % 74520 75943 22352 -1783954998 -1783954972
% L13:60 % 26 104 -1783954986 600 -13
% L13:65 % 100 -1300 337257256 337257164 12
% L13:70 % 1941920104 11 118 3001900 20590662
% L13:75 % 17067280 60 100 1189189975 8
% L13:80 % 24 74 592 7 2235246
% L13:85 % 55308 369 371 0 75916
% L13:90 % 74521 5 34787 5 1189190021
% L13:95 % 10 66272723 0 1189191411 89394
% L13:100 % 2147483647 6 900 14 160989
% L13:105 % 89394 31 2099392 4691 2099386
% L13:110 % 6 100 50 1938587407 1941919883
% L13:115 % 1941919909 26 13 1941919896 26
% L13:120 % 14 13367 50 100 10
% L13:125 % 0 1941920104 2147483647 3276500 3387810
% L13:130 % 2 2 0 99 0
% L13:135 % 0 0 55308 5 70
% L13:140 % 0 5 36 50 50
% L13:145 % 294745 5 5 5 26
% L13:150 % 12 20 516900 -516900 3332502
% L13:155 % 0 -10 0 0 4589052
% L13:160 % 23 29 24 1220 45
% L13:165 % 1941920124 1941921136 1941920124 1941921136 6706
% L13:170 % 12817 18417 1382 600 800
% L13:175 % 4 4 42 23 38
% L13:180 % 337267011 70 51434 1000000 371000000
% L13:185 % 1 1 337266996 71 51308
% L13:190 % 369000000 0 0 0 0
DATA L19
% L19:0 % 1188992105 1189171279 1189189703 1173491918 1173492124
% L19:5 % 1173492327 1173492532 1173492737 1173492942 1173493146
% L19:10 % 1173493350 1173493558 1173490278 1173490483 1173490688
% L19:15 % 1173490894 1173491098 0 0 0
DATA L20
% L20:0 % 1177003999 1177037277 1177037787 1177111741 1177113276
% L20:5 % 1188992406 1189027506 1189029039 1189171575 1189189992
% L20:10 % 1173712384 1173712409 1173712436 1173712469 1173712496
% L20:15 % 1173712523 1173712551 1173712573 1173712597 1173712622
% L20:20 % 1173712644 1173712667 1173712698 1173712723 1173713158
% L20:25 % 1173713183 1173713205 1173713230 1173713259 1173713288
% L20:30 % 1173713315 1173713344 1173713365 1173713391 1173713423
% L20:35 % 1173713445 1173713474 1173713495 1173713526 1173713547
% L20:40 % 1173713974 1173714001 1173714025 1173714081 1173714136
% L20:45 % 1173714198 1173714245 1173714294 1173714348 1177002452
DATA L21
% L21:0 % 1941096388 1941120530 1941120899 1941174579 1941175694
% L21:5 % 1941776718 1941802193 1941803306 1941906757 1941920124
% L21:10 % 1938419405 1938419419 1938419434 1938419452 1938419467
% L21:15 % 1938419482 1938419498 1938419510 1938419523 1938419537
% L21:20 % 1938419549 1938419562 1938419579 1938419593 1938419834
% L21:25 % 1938419848 1938419860 1938419874 1938419890 1938419906
% L21:30 % 1938419921 1938419937 1938419949 1938419963 1938419981
% L21:35 % 1938419993 1938420009 1938420021 1938420038 1938420050
% L21:40 % 1938420287 1938420302 1938420315 1938420346 1938420377
% L21:45 % 1938420411 1938420437 1938420464 1938420494 1941095259
DATA L22
% L22:0 % 1177040119 1177040629 1177111819 1177112335 1177112845
% L22:5 % 1177113358 1177113875 1188992414 1188993767 1189027580
% L22:10 % 1189029107 1189171589 1189190005 1189191387 1097515193
% L22:15 % 1097515421 1164146194 1164182576 1164198280 1164198510
% L22:20 % 1164198739 1164198968 1164223426 1164253092 1164262458
% L22:25 % 1164336774 1164344878 1164357608 1164367350 1164385327
% L22:30 % 1164400986 1164407890 1164419585 1164427785 1164433444
% L22:35 % 1164439941 1164463880 1164479155 1172337748 1172366635
% L22:40 % 1172382490 1172446970 1172844337 1172867913 1172898737
% L22:45 % 1173009549 1173016946 1173136175 1177002543 1177004082
DATA L23
% L23:0 % 1941122592 1941122963 1941174636 1941175010 1941175381
% L23:5 % 1941175754 1941176129 1941776724 1941777706 1941802247
% L23:10 % 1941803355 1941906767 1941920134 1941921136 1923690900
% L23:15 % 1923690969 1933152542 1933172714 1933181421 1933181549
% L23:20 % 1933181676 1933181802 1933195362 1933211809 1933217001
% L23:25 % 1933258208 1933262699 1933269756 1933275158 1933285125
% L23:30 % 1933293808 1933297636 1933304120 1933308667 1933311804
% L23:35 % 1933315405 1933328677 1933337146 1937694172 1937710185
% L23:40 % 1937718977 1937754728 1937975041 1937988112 1938005198
% L23:45 % 1938066636 1938070737 1938136840 1941095326 1941096448
DATA L30
% L30:0 % 1097513510 1097513738 1097513967 1097514196 1097514426
% L30:5 % 1097514655 1097514883 1097515111 1097515339 1188692931
% L30:10 % 1071304952 1071305179 1071305406 1071305631 1071305859
% L30:15 % 1071306086 1071306312 1071306539 1071306765 1071306992
% L30:20 % 1071307217 1071307442 1071307668 1071307895 1071308121
% L30:25 % 1071308347 1071308573 1071308799 1071309024 1071309250
% L30:30 % 1071309476 1071429569 1071429795 1071431153 1071431379
% L30:35 % 1071431606 1088333039 1088333266 1088334623 1088334848
% L30:40 % 1088335075 1089808842 1089809070 1089810430 1089810657
% L30:45 % 1089810882 1092780028 1092791426 1092806921 1097513283
DATA L31
% L31:0 % 3522828 3522897 3522967 3523035 3523105
% L31:5 % 3523175 3523244 3523313 3523382 20590662
% L31:10 % 2077757 2077757 2077757 2077757 2077757
% L31:15 % 2077757 2077757 2077757 2077757 2077757
% L31:20 % 2077757 2077757 2077757 2077757 2077757
% L31:25 % 2077757 2077757 2077757 2077757 2077757
% L31:30 % 2077757 2077757 2077757 2077757 2077757
% L31:35 % 2077757 2077757 2077757 2077757 2077757
% L31:40 % 2077757 2077757 2077757 2077757 2077757
% L31:45 % 2077757 2091375 2094821 2099507 3522760
DATA L32
% L32:0 % 1186638188 1186638693 1186639199 1186639703 1186640207
% L32:5 % 1186640711 1186641217 1186641721 1188691063 1188992386
% L32:10 % 1189027435 1189028975 1189189964 1186619532 1186620036
% L32:15 % 1186620541 1186621044 1186621549 1186622052 1186622555
% L32:20 % 1186623059 1186623563 1186624069 1186624573 1186625077
% L32:25 % 1186625582 1186626085 1186626589 1186627093 1186627598
% L32:30 % 1186628101 1186628604 1186629110 1186629615 1186630120
% L32:35 % 1186630624 1186631128 1186631633 1186632137 1186632642
% L32:40 % 1186633147 1186633651 1186634155 1186634659 1186635164
% L32:45 % 1186635668 1186636171 1186636676 1186637181 1186637685
DATA L33
% L33:0 % 1941353968 1941353968 1941353968 1941353968 1941353968
% L33:5 % 1941353968 1941353968 1941353968 1941743022 1941776703
% L33:10 % 1941802142 1941803259 1941920104 1941353968 1941353968
% L33:15 % 1941353968 1941353968 1941353968 1941353968 1941353968
% L33:20 % 1941353968 1941353968 1941353968 1941353968 1941353968
% L33:25 % 1941353968 1941353968 1941353968 1941353968 1941353968
% L33:30 % 1941353968 1941353968 1941353968 1941353968 1941353968
% L33:35 % 1941353968 1941353968 1941353968 1941353968 1941353968
% L33:40 % 1941353968 1941353968 1941353968 1941353968 1941353968
% L33:45 % 1941353968 1941353968 1941353968 1941353968 1941353968
DATA B38
% B38:0 % 0X0100
DATA B100
% B100:0 % 0X2780 0X18A8 0X0004 0X0000 0X0000 0X0000 0X0000 0X0000 0X0000 0X0000
DATA N101
% N101:0 % 118 0 0 0 1183 100 1002 1200 1210 1230
% N101:10 % 1240 1600 10 16383 1269 17365 3043 500 333 500
% N101:20 % 1000 500 400 0 0 0 500 500 0 0
DATA L102
% L102:0 % 40 10 7213 7192 7200
% L102:5 % 7200 1 1 0 0
% L102:10 % -516900 1 0 0 34787
% L102:15 % 0 30 10 30 10
% L102:20 % 0 6 71085 0 29
% L102:25 % 33 0 91177564 81649 32
% L102:30 % 11 0 9 7730 0
% L102:35 % 174 302 0 999999 24
% L102:40 % 1 8 0 1 0
